(* Logix 5000 project; controller Receptivo vendor 1 type 14 code 106 rev 30.11; software revision 30.00; part 6 of 10 *)
(* tags used below, declared in another part *)
   Codigo_QAD3_Espacios : DINT;
   Codigo_QAD4_Espacios : DINT;
   Descripcion3_Espacios : DINT;
   Descripcion4_Espacios : DINT;
   Numero_Espacios_Descripcion_3 : DINT;
   Numero_Espacios_Descripcion_4 : DINT;
   Numero_Espacios_QAD3 : DINT;
   Numero_Espacios_QAD4 : DINT;
   Print3_Ejecute : BOOL;
   Print3_OK : BOOL;
   Print4_Ejecute : BOOL;
   Print4_OK : BOOL;
   CAJAS_3 : DINT;
   CAJAS_4 : DINT;
   Calendario : Hora_y_Fecha;
   CERO : DINT;
   Clima_3 : DINT;
   Clima_4 : DINT;
   Consecutivo : INT;
   Densidad_3 : REAL;
   Densidad_4 : REAL;
   Densidad_Bidon : REAL;
   Densidad_Bidon_1 : REAL;
   Densidad_Elmar_1 : REAL;
   Densidad_Fogg1_1 : REAL;
   Densidad_Fogg2_1 : REAL;
   EAN14_3 : Codigo_Barras;
   EAN14_4 : Codigo_Barras;
   Espacios : STRING;
   Estacion_1_GCola_1 : UDT_COLA;
   Estacion_1_General : UDT_GENERAL;
   Estacion_2_GCola_1 : UDT_COLA;
   ESTACION_3 : DINT;
   Estacion_3_GCola_1 : UDT_COLA;
   Estacion_3_General : UDT_GENERAL;
   Estacion_3_String : STRING;
   ESTACION_4 : DINT;
   Estacion_4_GCola_1 : UDT_COLA;
   Estacion_4_General : UDT_GENERAL;
   Estacion_4_String : STRING;
   LInea_General_3 : INT;
   LInea_General_4 : INT;
   Linea_String_General : STRING;
   Lote : DINT;
   Operador_3 : DINT;
   Operador_4 : DINT;
   Pesaje_3 : REAL;
   Pesaje_4 : REAL;
   Peso_Bidones : REAL;
   Peso_Bidones_1 : REAL;
   Peso_Caja_Elmar_1 : REAL;
   Peso_Caja_Fogg1_1 : REAL;
   Peso_Caja_Fogg2_1 : REAL;
   PESO_REAL_3 : DINT;
   PESO_REAL_4 : DINT;
   PESO_TEORICO_3 : DINT;
   PESO_TEORICO_4 : DINT;
   Producido_Bidones_Ahora : UDT_Maestro;
   Producido_Elmar_Ahora : UDT_Maestro;
   Producido_Fogg1_Ahora : UDT_Maestro;
   Producido_Fogg2_Ahora : UDT_Maestro;
   Producto3 : UDT_Inventario;
   Producto4 : UDT_Inventario;
   QAD_3 : STRING;
   QAD_4 : STRING;
   QAD_Auxiliar_Est4 : STRING;
(* MainProgram, continued *)

ROUTINE Estacion_3_Datos   (* ladder *)
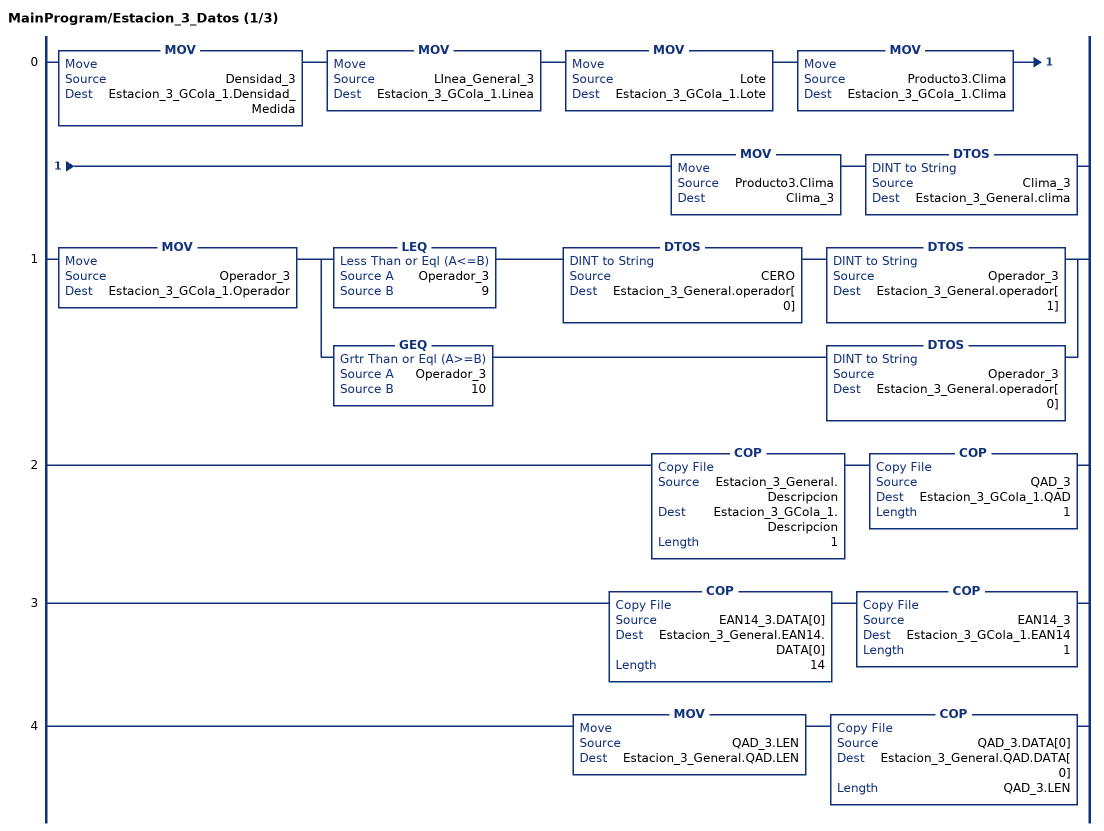
   0: MOV(Densidad_3,Estacion_3_GCola_1.Densidad_Medida)MOV(LInea_General_3,Estacion_3_GCola_1.Linea)MOV(Lote,Estacion_3_GCola_1.Lote)MOV(Producto3.Clima,Estacion_3_GCola_1.Clima)MOV(Producto3.Clima,Clima_3)DTOS(Clima_3,Estacion_3_General.clima);
   1: MOV(Operador_3,Estacion_3_GCola_1.Operador)[LEQ(Operador_3,9) DTOS(CERO,Estacion_3_General.operador[0]) DTOS(Operador_3,Estacion_3_General.operador[1]) ,GEQ(Operador_3,10) DTOS(Operador_3,Estacion_3_General.operador[0]) ];
   2: COP(Estacion_3_General.Descripcion,Estacion_3_GCola_1.Descripcion,1)COP(QAD_3,Estacion_3_GCola_1.QAD,1);
   3: COP(EAN14_3.DATA[0],Estacion_3_General.EAN14.DATA[0],14)COP(EAN14_3,Estacion_3_GCola_1.EAN14,1);
   4: MOV(QAD_3.LEN,Estacion_3_General.QAD.LEN)COP(QAD_3.DATA[0],Estacion_3_General.QAD.DATA[0],QAD_3.LEN);
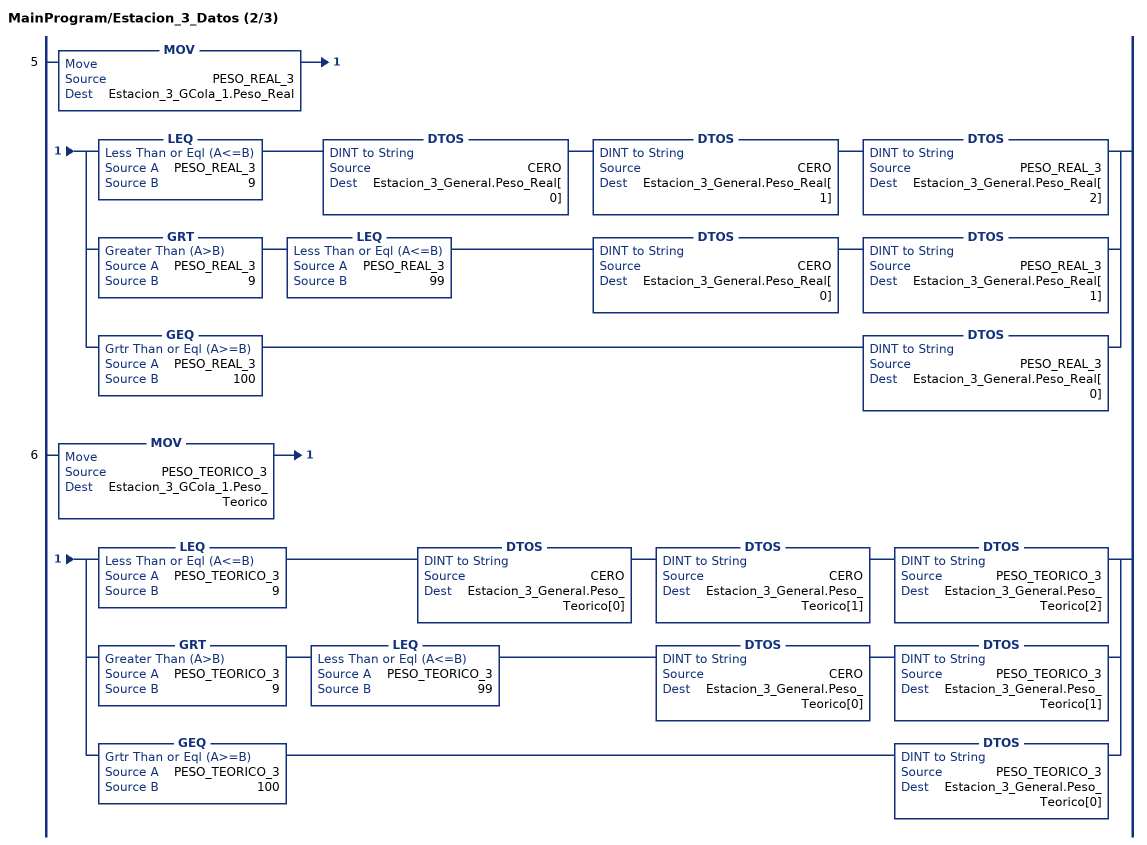
   5: MOV(PESO_REAL_3,Estacion_3_GCola_1.Peso_Real)[LEQ(PESO_REAL_3,9) DTOS(CERO,Estacion_3_General.Peso_Real[0]) DTOS(CERO,Estacion_3_General.Peso_Real[1]) DTOS(PESO_REAL_3,Estacion_3_General.Peso_Real[2]) ,GRT(PESO_REAL_3,9) LEQ(PESO_REAL_3,99) DTOS(CERO,Estacion_3_General.Peso_Real[0]) DTOS(PESO_REAL_3,Estacion_3_General.Peso_Real[1]) ,GEQ(PESO_REAL_3,100) DTOS(PESO_REAL_3,Estacion_3_General.Peso_Real[0]) ];
   6: MOV(PESO_TEORICO_3,Estacion_3_GCola_1.Peso_Teorico)[LEQ(PESO_TEORICO_3,9) DTOS(CERO,Estacion_3_General.Peso_Teorico[0]) DTOS(CERO,Estacion_3_General.Peso_Teorico[1]) DTOS(PESO_TEORICO_3,Estacion_3_General.Peso_Teorico[2]) ,GRT(PESO_TEORICO_3,9) LEQ(PESO_TEORICO_3,99) DTOS(CERO,Estacion_3_General.Peso_Teorico[0]) DTOS(PESO_TEORICO_3,Estacion_3_General.Peso_Teorico[1]) ,GEQ(PESO_TEORICO_3,100) DTOS(PESO_TEORICO_3,Estacion_3_General.Peso_Teorico[0]) ];
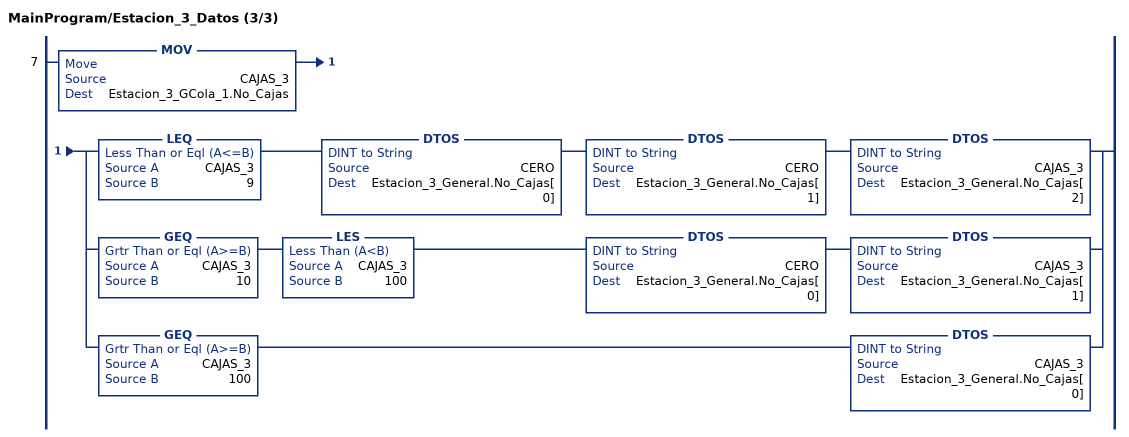
   7: MOV(CAJAS_3,Estacion_3_GCola_1.No_Cajas)[LEQ(CAJAS_3,9) DTOS(CERO,Estacion_3_General.No_Cajas[0]) DTOS(CERO,Estacion_3_General.No_Cajas[1]) DTOS(CAJAS_3,Estacion_3_General.No_Cajas[2]) ,GEQ(CAJAS_3,10) LES(CAJAS_3,100) DTOS(CERO,Estacion_3_General.No_Cajas[0]) DTOS(CAJAS_3,Estacion_3_General.No_Cajas[1]) ,GEQ(CAJAS_3,100) DTOS(CAJAS_3,Estacion_3_General.No_Cajas[0]) ];
END_ROUTINE

ROUTINE Estacion_3_To_Printer   (* ladder *)
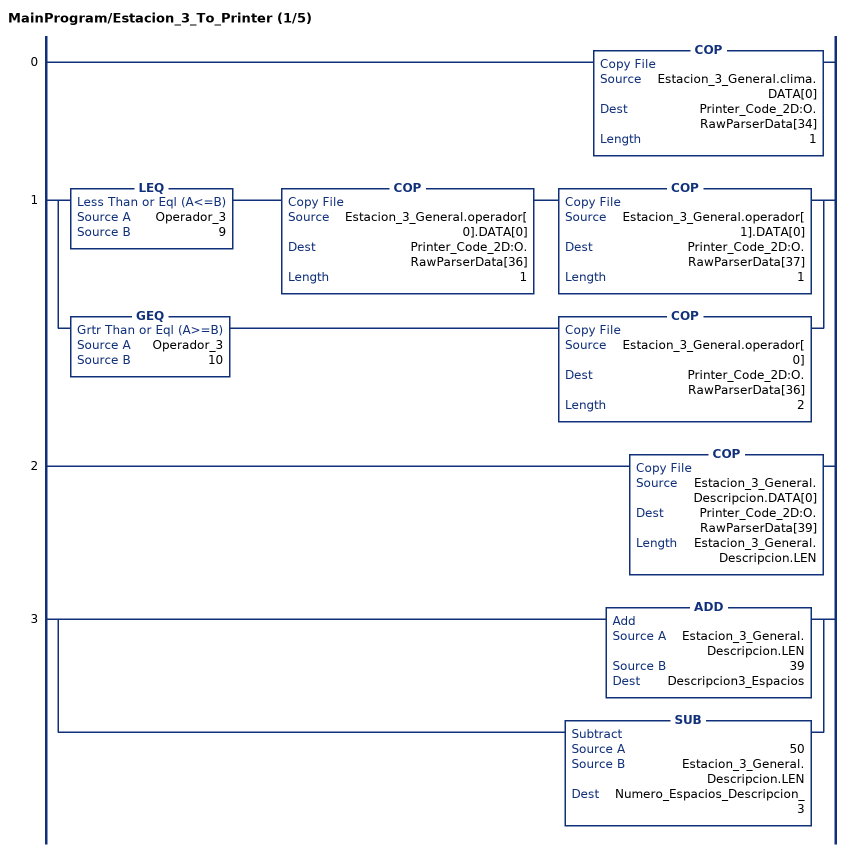
   0: COP(Estacion_3_General.clima.DATA[0],Printer_Code_2D:O.RawParserData[34],1);
   1: [LEQ(Operador_3,9) COP(Estacion_3_General.operador[0].DATA[0],Printer_Code_2D:O.RawParserData[36],1) COP(Estacion_3_General.operador[1].DATA[0],Printer_Code_2D:O.RawParserData[37],1) ,GEQ(Operador_3,10) COP(Estacion_3_General.operador[0],Printer_Code_2D:O.RawParserData[36],2) ];
   2: COP(Estacion_3_General.Descripcion.DATA[0],Printer_Code_2D:O.RawParserData[39],Estacion_3_General.Descripcion.LEN);
   3: [ADD(Estacion_3_General.Descripcion.LEN,39,Descripcion3_Espacios) ,SUB(50,Estacion_3_General.Descripcion.LEN,Numero_Espacios_Descripcion_3) ];
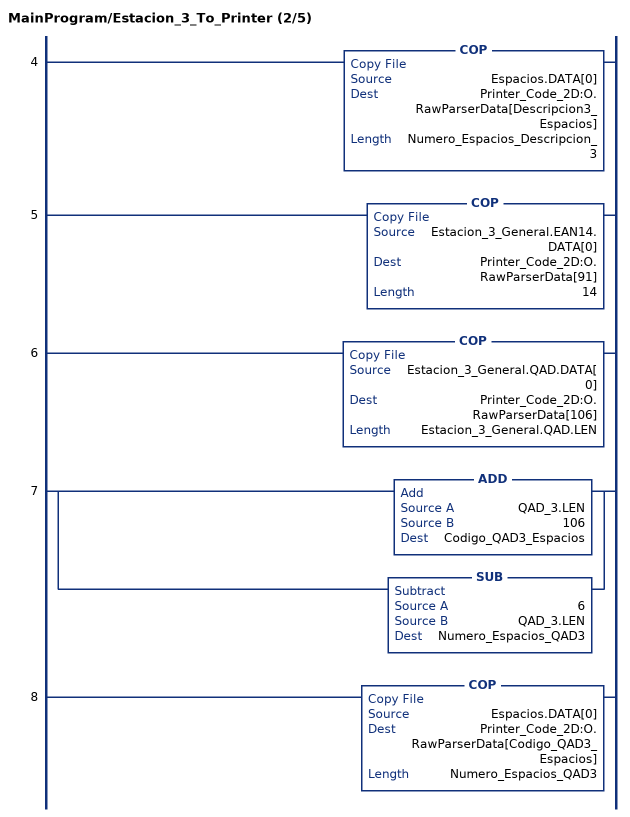
   4: COP(Espacios.DATA[0],Printer_Code_2D:O.RawParserData[Descripcion3_Espacios],Numero_Espacios_Descripcion_3);
   5: COP(Estacion_3_General.EAN14.DATA[0],Printer_Code_2D:O.RawParserData[91],14);
   6: COP(Estacion_3_General.QAD.DATA[0],Printer_Code_2D:O.RawParserData[106],Estacion_3_General.QAD.LEN);
   7: [ADD(QAD_3.LEN,106,Codigo_QAD3_Espacios) ,SUB(6,QAD_3.LEN,Numero_Espacios_QAD3) ];
   8: COP(Espacios.DATA[0],Printer_Code_2D:O.RawParserData[Codigo_QAD3_Espacios],Numero_Espacios_QAD3);
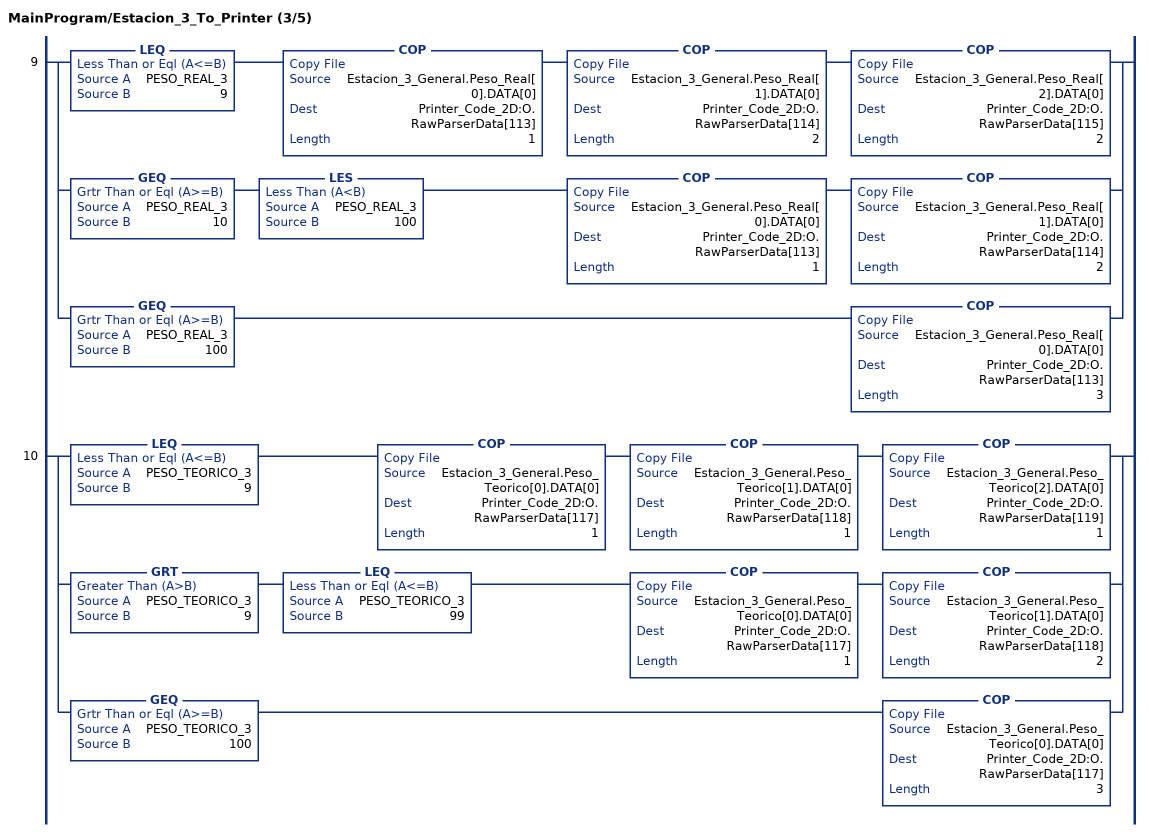
   9: [LEQ(PESO_REAL_3,9) COP(Estacion_3_General.Peso_Real[0].DATA[0],Printer_Code_2D:O.RawParserData[113],1) COP(Estacion_3_General.Peso_Real[1].DATA[0],Printer_Code_2D:O.RawParserData[114],2) COP(Estacion_3_General.Peso_Real[2].DATA[0],Printer_Code_2D:O.RawParserData[115],2) ,GEQ(PESO_REAL_3,10) LES(PESO_REAL_3,100) COP(Estacion_3_General.Peso_Real[0].DATA[0],Printer_Code_2D:O.RawParserData[113],1) COP(Estacion_3_General.Peso_Real[1].DATA[0],Printer_Code_2D:O.RawParserData[114],2) ,GEQ(PESO_REAL_3,100) COP(Estacion_3_General.Peso_Real[0].DATA[0],Printer_Code_2D:O.RawParserData[113],3) ];
   10: [LEQ(PESO_TEORICO_3,9) COP(Estacion_3_General.Peso_Teorico[0].DATA[0],Printer_Code_2D:O.RawParserData[117],1) COP(Estacion_3_General.Peso_Teorico[1].DATA[0],Printer_Code_2D:O.RawParserData[118],1) COP(Estacion_3_General.Peso_Teorico[2].DATA[0],Printer_Code_2D:O.RawParserData[119],1) ,GRT(PESO_TEORICO_3,9) LEQ(PESO_TEORICO_3,99) COP(Estacion_3_General.Peso_Teorico[0].DATA[0],Printer_Code_2D:O.RawParserData[117],1) COP(Estacion_3_General.Peso_Teorico[1].DATA[0],Printer_Code_2D:O.RawParserData[118],2) ,GEQ(PESO_TEORICO_3,100) COP(Estacion_3_General.Peso_Teorico[0].DATA[0],Printer_Code_2D:O.RawParserData[117],3) ];
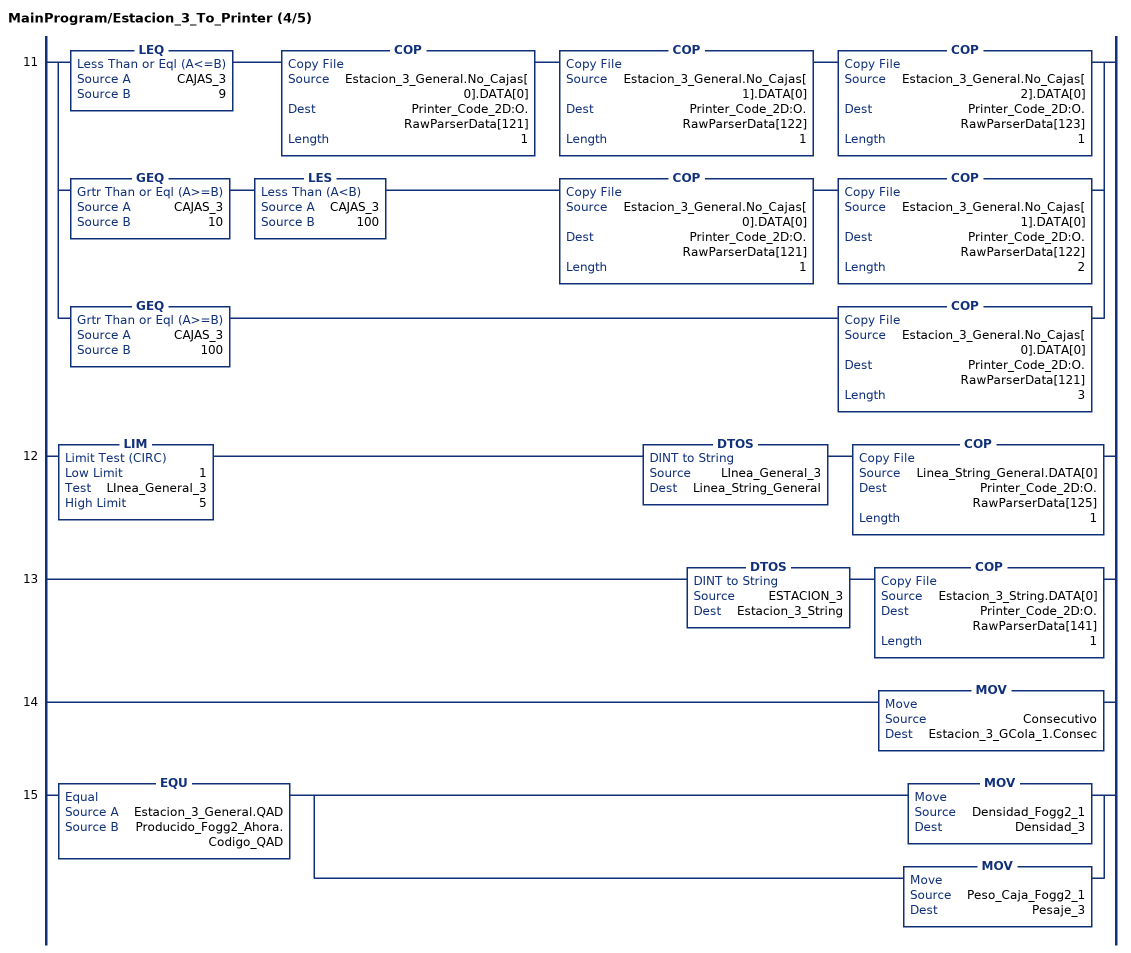
   11: [LEQ(CAJAS_3,9) COP(Estacion_3_General.No_Cajas[0].DATA[0],Printer_Code_2D:O.RawParserData[121],1) COP(Estacion_3_General.No_Cajas[1].DATA[0],Printer_Code_2D:O.RawParserData[122],1) COP(Estacion_3_General.No_Cajas[2].DATA[0],Printer_Code_2D:O.RawParserData[123],1) ,GEQ(CAJAS_3,10) LES(CAJAS_3,100) COP(Estacion_3_General.No_Cajas[0].DATA[0],Printer_Code_2D:O.RawParserData[121],1) COP(Estacion_3_General.No_Cajas[1].DATA[0],Printer_Code_2D:O.RawParserData[122],2) ,GEQ(CAJAS_3,100) COP(Estacion_3_General.No_Cajas[0].DATA[0],Printer_Code_2D:O.RawParserData[121],3) ];
   12: LIM(1,LInea_General_3,5)DTOS(LInea_General_3,Linea_String_General)COP(Linea_String_General.DATA[0],Printer_Code_2D:O.RawParserData[125],1);
   13: DTOS(ESTACION_3,Estacion_3_String)COP(Estacion_3_String.DATA[0],Printer_Code_2D:O.RawParserData[141],1);
   14: MOV(Consecutivo,Estacion_3_GCola_1.Consec);
   15: EQU(Estacion_3_General.QAD,Producido_Fogg2_Ahora.Codigo_QAD)[MOV(Densidad_Fogg2_1,Densidad_3) ,MOV(Peso_Caja_Fogg2_1,Pesaje_3) ];
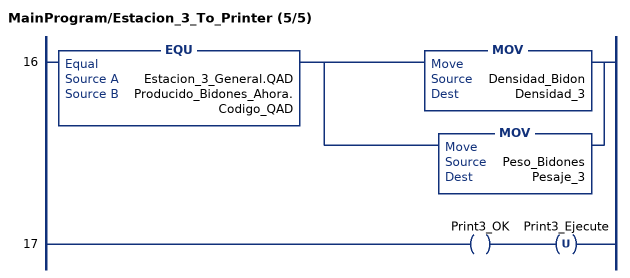
   16: EQU(Estacion_3_General.QAD,Producido_Bidones_Ahora.Codigo_QAD)[MOV(Densidad_Bidon,Densidad_3) ,MOV(Peso_Bidones,Pesaje_3) ];
   17: OTE(Print3_OK)OTU(Print3_Ejecute);
END_ROUTINE

ROUTINE Estacion_4_Datos   (* ladder *)
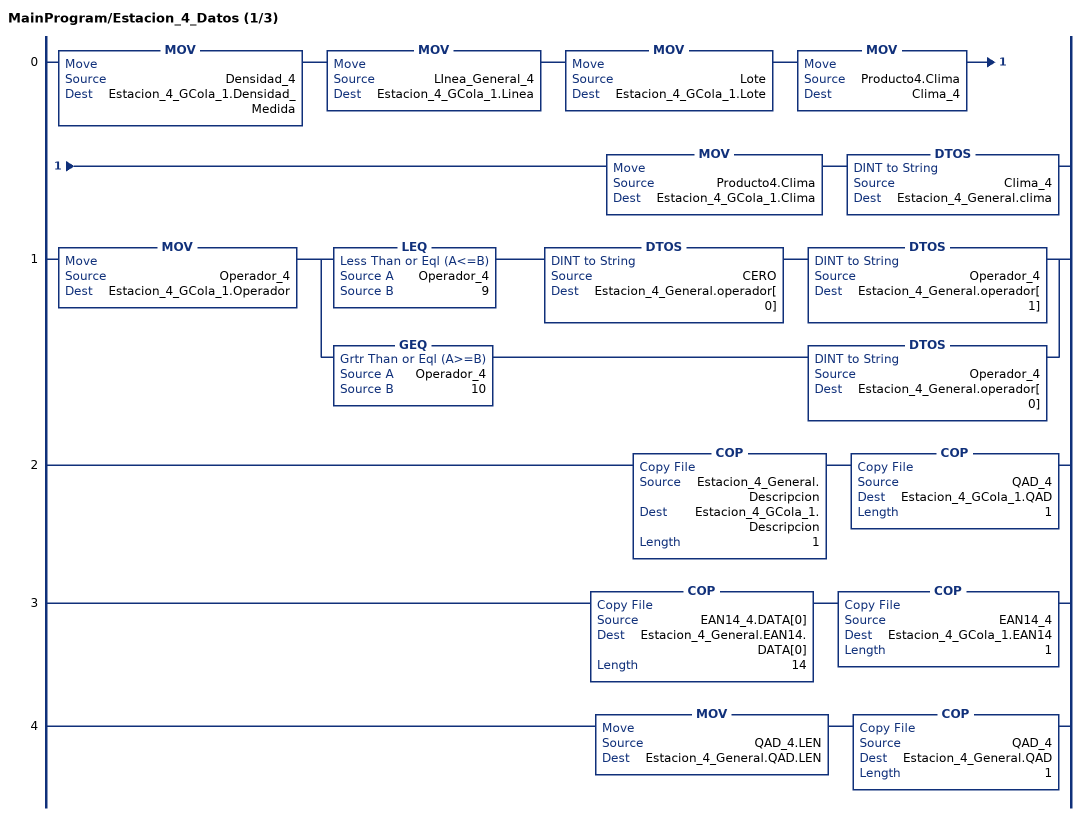
   0: MOV(Densidad_4,Estacion_4_GCola_1.Densidad_Medida)MOV(LInea_General_4,Estacion_4_GCola_1.Linea)MOV(Lote,Estacion_4_GCola_1.Lote)MOV(Producto4.Clima,Clima_4)MOV(Producto4.Clima,Estacion_4_GCola_1.Clima)DTOS(Clima_4,Estacion_4_General.clima);
   1: MOV(Operador_4,Estacion_4_GCola_1.Operador)[LEQ(Operador_4,9) DTOS(CERO,Estacion_4_General.operador[0]) DTOS(Operador_4,Estacion_4_General.operador[1]) ,GEQ(Operador_4,10) DTOS(Operador_4,Estacion_4_General.operador[0]) ];
   2: COP(Estacion_4_General.Descripcion,Estacion_4_GCola_1.Descripcion,1)COP(QAD_4,Estacion_4_GCola_1.QAD,1);
   3: COP(EAN14_4.DATA[0],Estacion_4_General.EAN14.DATA[0],14)COP(EAN14_4,Estacion_4_GCola_1.EAN14,1);
   4: MOV(QAD_4.LEN,Estacion_4_General.QAD.LEN)COP(QAD_4,Estacion_4_General.QAD,1);
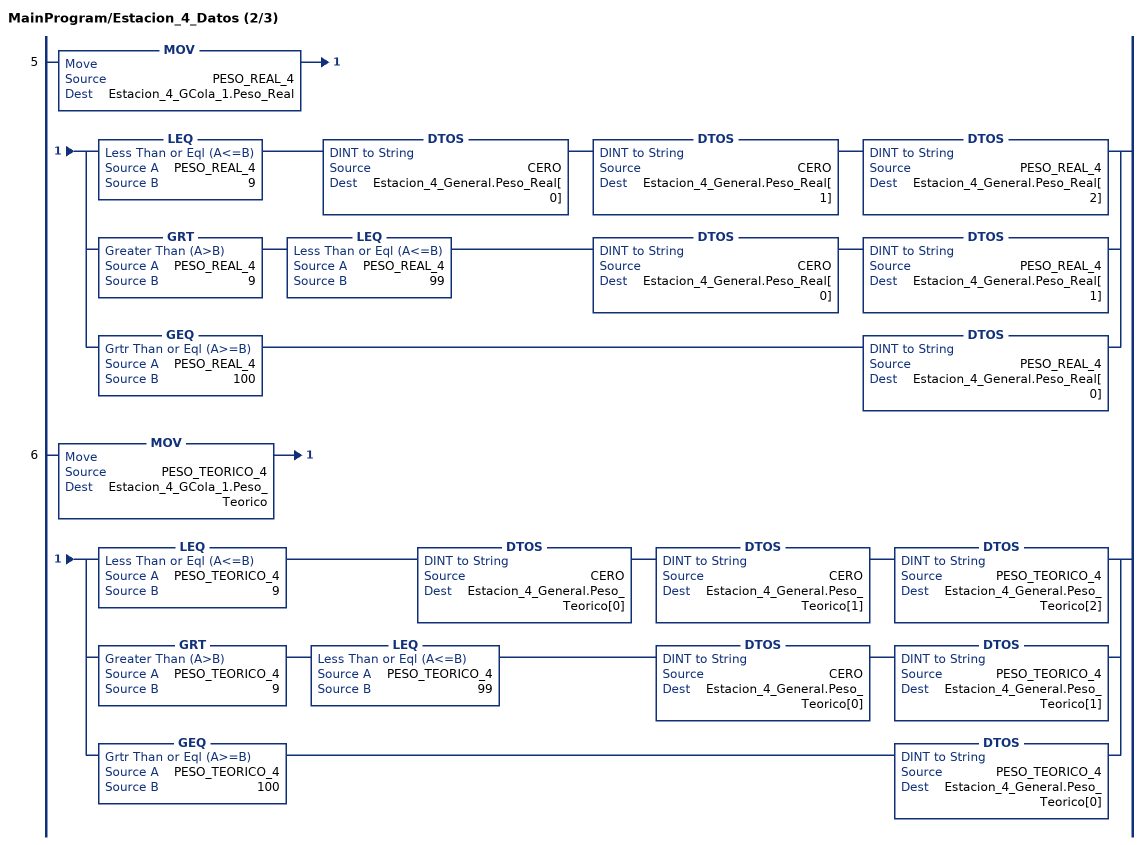
   5: MOV(PESO_REAL_4,Estacion_4_GCola_1.Peso_Real)[LEQ(PESO_REAL_4,9) DTOS(CERO,Estacion_4_General.Peso_Real[0]) DTOS(CERO,Estacion_4_General.Peso_Real[1]) DTOS(PESO_REAL_4,Estacion_4_General.Peso_Real[2]) ,GRT(PESO_REAL_4,9) LEQ(PESO_REAL_4,99) DTOS(CERO,Estacion_4_General.Peso_Real[0]) DTOS(PESO_REAL_4,Estacion_4_General.Peso_Real[1]) ,GEQ(PESO_REAL_4,100) DTOS(PESO_REAL_4,Estacion_4_General.Peso_Real[0]) ];
   6: MOV(PESO_TEORICO_4,Estacion_4_GCola_1.Peso_Teorico)[LEQ(PESO_TEORICO_4,9) DTOS(CERO,Estacion_4_General.Peso_Teorico[0]) DTOS(CERO,Estacion_4_General.Peso_Teorico[1]) DTOS(PESO_TEORICO_4,Estacion_4_General.Peso_Teorico[2]) ,GRT(PESO_TEORICO_4,9) LEQ(PESO_TEORICO_4,99) DTOS(CERO,Estacion_4_General.Peso_Teorico[0]) DTOS(PESO_TEORICO_4,Estacion_4_General.Peso_Teorico[1]) ,GEQ(PESO_TEORICO_4,100) DTOS(PESO_TEORICO_4,Estacion_4_General.Peso_Teorico[0]) ];
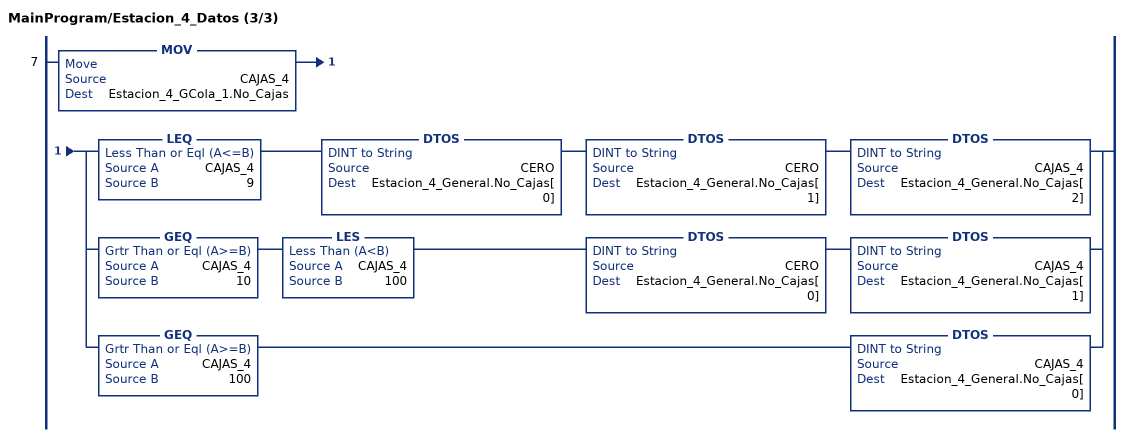
   7: MOV(CAJAS_4,Estacion_4_GCola_1.No_Cajas)[LEQ(CAJAS_4,9) DTOS(CERO,Estacion_4_General.No_Cajas[0]) DTOS(CERO,Estacion_4_General.No_Cajas[1]) DTOS(CAJAS_4,Estacion_4_General.No_Cajas[2]) ,GEQ(CAJAS_4,10) LES(CAJAS_4,100) DTOS(CERO,Estacion_4_General.No_Cajas[0]) DTOS(CAJAS_4,Estacion_4_General.No_Cajas[1]) ,GEQ(CAJAS_4,100) DTOS(CAJAS_4,Estacion_4_General.No_Cajas[0]) ];
END_ROUTINE

ROUTINE Estacion_4_To_Printer   (* ladder *)
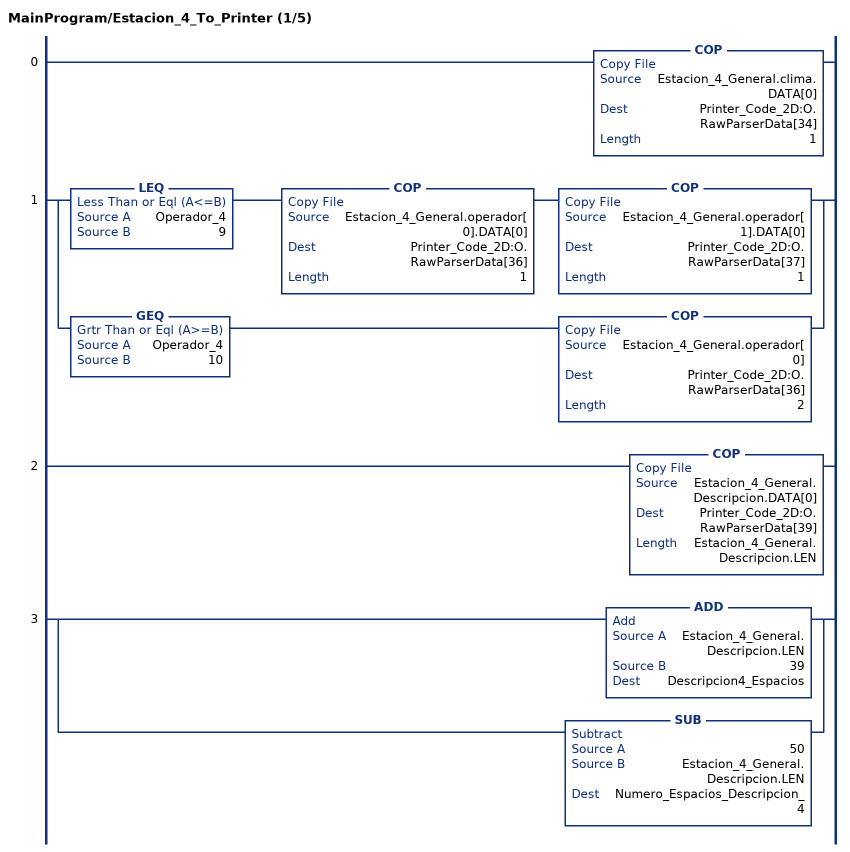
   0: COP(Estacion_4_General.clima.DATA[0],Printer_Code_2D:O.RawParserData[34],1);
   1: [LEQ(Operador_4,9) COP(Estacion_4_General.operador[0].DATA[0],Printer_Code_2D:O.RawParserData[36],1) COP(Estacion_4_General.operador[1].DATA[0],Printer_Code_2D:O.RawParserData[37],1) ,GEQ(Operador_4,10) COP(Estacion_4_General.operador[0],Printer_Code_2D:O.RawParserData[36],2) ];
   2: COP(Estacion_4_General.Descripcion.DATA[0],Printer_Code_2D:O.RawParserData[39],Estacion_4_General.Descripcion.LEN);
   3: [ADD(Estacion_4_General.Descripcion.LEN,39,Descripcion4_Espacios) ,SUB(50,Estacion_4_General.Descripcion.LEN,Numero_Espacios_Descripcion_4) ];
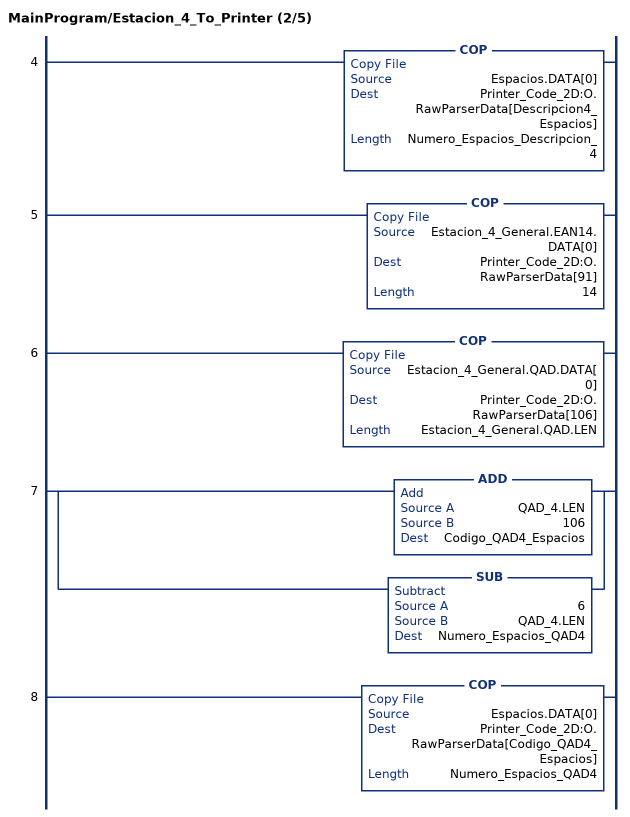
   4: COP(Espacios.DATA[0],Printer_Code_2D:O.RawParserData[Descripcion4_Espacios],Numero_Espacios_Descripcion_4);
   5: COP(Estacion_4_General.EAN14.DATA[0],Printer_Code_2D:O.RawParserData[91],14);
   6: COP(Estacion_4_General.QAD.DATA[0],Printer_Code_2D:O.RawParserData[106],Estacion_4_General.QAD.LEN);
   7: [ADD(QAD_4.LEN,106,Codigo_QAD4_Espacios) ,SUB(6,QAD_4.LEN,Numero_Espacios_QAD4) ];
   8: COP(Espacios.DATA[0],Printer_Code_2D:O.RawParserData[Codigo_QAD4_Espacios],Numero_Espacios_QAD4);
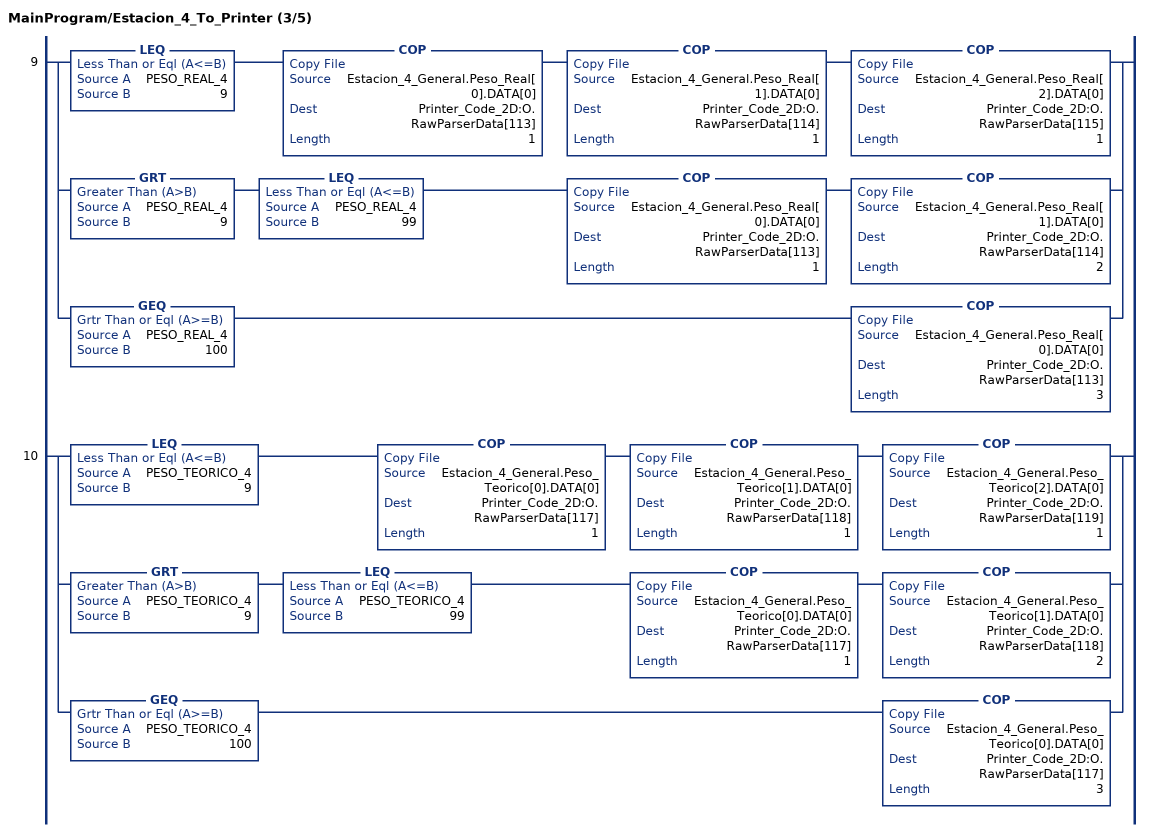
   9: [LEQ(PESO_REAL_4,9) COP(Estacion_4_General.Peso_Real[0].DATA[0],Printer_Code_2D:O.RawParserData[113],1) COP(Estacion_4_General.Peso_Real[1].DATA[0],Printer_Code_2D:O.RawParserData[114],1) COP(Estacion_4_General.Peso_Real[2].DATA[0],Printer_Code_2D:O.RawParserData[115],1) ,GRT(PESO_REAL_4,9) LEQ(PESO_REAL_4,99) COP(Estacion_4_General.Peso_Real[0].DATA[0],Printer_Code_2D:O.RawParserData[113],1) COP(Estacion_4_General.Peso_Real[1].DATA[0],Printer_Code_2D:O.RawParserData[114],2) ,GEQ(PESO_REAL_4,100) COP(Estacion_4_General.Peso_Real[0].DATA[0],Printer_Code_2D:O.RawParserData[113],3) ];
   10: [LEQ(PESO_TEORICO_4,9) COP(Estacion_4_General.Peso_Teorico[0].DATA[0],Printer_Code_2D:O.RawParserData[117],1) COP(Estacion_4_General.Peso_Teorico[1].DATA[0],Printer_Code_2D:O.RawParserData[118],1) COP(Estacion_4_General.Peso_Teorico[2].DATA[0],Printer_Code_2D:O.RawParserData[119],1) ,GRT(PESO_TEORICO_4,9) LEQ(PESO_TEORICO_4,99) COP(Estacion_4_General.Peso_Teorico[0].DATA[0],Printer_Code_2D:O.RawParserData[117],1) COP(Estacion_4_General.Peso_Teorico[1].DATA[0],Printer_Code_2D:O.RawParserData[118],2) ,GEQ(PESO_TEORICO_4,100) COP(Estacion_4_General.Peso_Teorico[0].DATA[0],Printer_Code_2D:O.RawParserData[117],3) ];
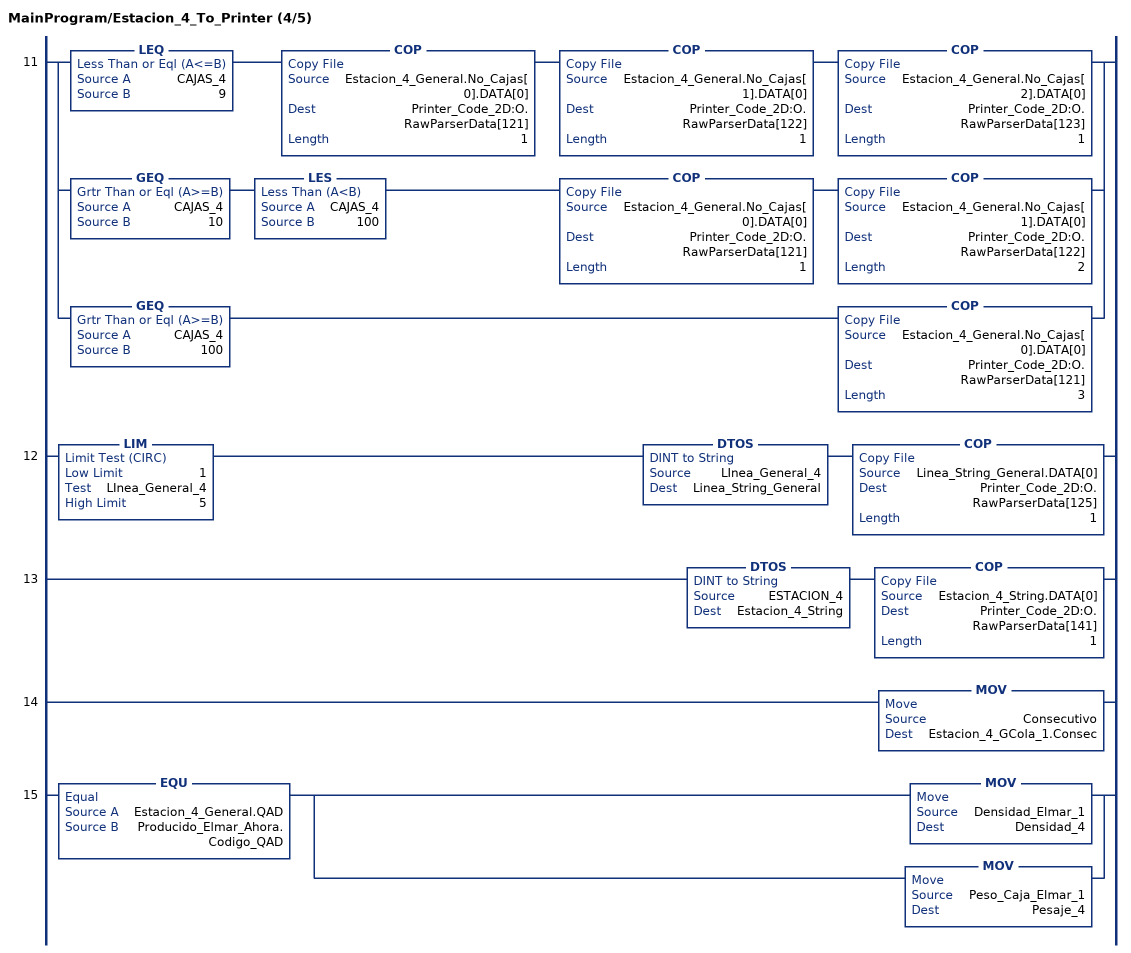
   11: [LEQ(CAJAS_4,9) COP(Estacion_4_General.No_Cajas[0].DATA[0],Printer_Code_2D:O.RawParserData[121],1) COP(Estacion_4_General.No_Cajas[1].DATA[0],Printer_Code_2D:O.RawParserData[122],1) COP(Estacion_4_General.No_Cajas[2].DATA[0],Printer_Code_2D:O.RawParserData[123],1) ,GEQ(CAJAS_4,10) LES(CAJAS_4,100) COP(Estacion_4_General.No_Cajas[0].DATA[0],Printer_Code_2D:O.RawParserData[121],1) COP(Estacion_4_General.No_Cajas[1].DATA[0],Printer_Code_2D:O.RawParserData[122],2) ,GEQ(CAJAS_4,100) COP(Estacion_4_General.No_Cajas[0].DATA[0],Printer_Code_2D:O.RawParserData[121],3) ];
   12: LIM(1,LInea_General_4,5)DTOS(LInea_General_4,Linea_String_General)COP(Linea_String_General.DATA[0],Printer_Code_2D:O.RawParserData[125],1);
   13: DTOS(ESTACION_4,Estacion_4_String)COP(Estacion_4_String.DATA[0],Printer_Code_2D:O.RawParserData[141],1);
   14: MOV(Consecutivo,Estacion_4_GCola_1.Consec);
   15: EQU(Estacion_4_General.QAD,Producido_Elmar_Ahora.Codigo_QAD)[MOV(Densidad_Elmar_1,Densidad_4) ,MOV(Peso_Caja_Elmar_1,Pesaje_4) ];
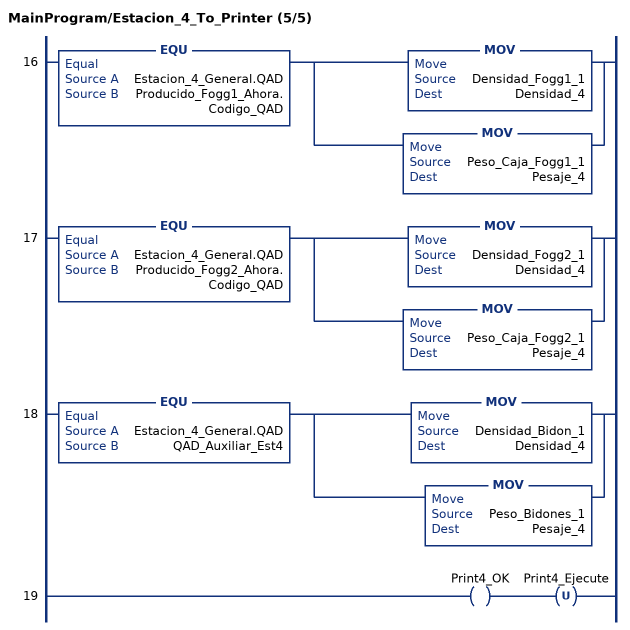
   16: EQU(Estacion_4_General.QAD,Producido_Fogg1_Ahora.Codigo_QAD)[MOV(Densidad_Fogg1_1,Densidad_4) ,MOV(Peso_Caja_Fogg1_1,Pesaje_4) ];
   17: EQU(Estacion_4_General.QAD,Producido_Fogg2_Ahora.Codigo_QAD)[MOV(Densidad_Fogg2_1,Densidad_4) ,MOV(Peso_Caja_Fogg2_1,Pesaje_4) ];
   18: EQU(Estacion_4_General.QAD,QAD_Auxiliar_Est4)[MOV(Densidad_Bidon_1,Densidad_4) ,MOV(Peso_Bidones_1,Pesaje_4) ];
   19: OTE(Print4_OK)OTU(Print4_Ejecute);
END_ROUTINE

ROUTINE Get_Date_Time   (* ladder *)
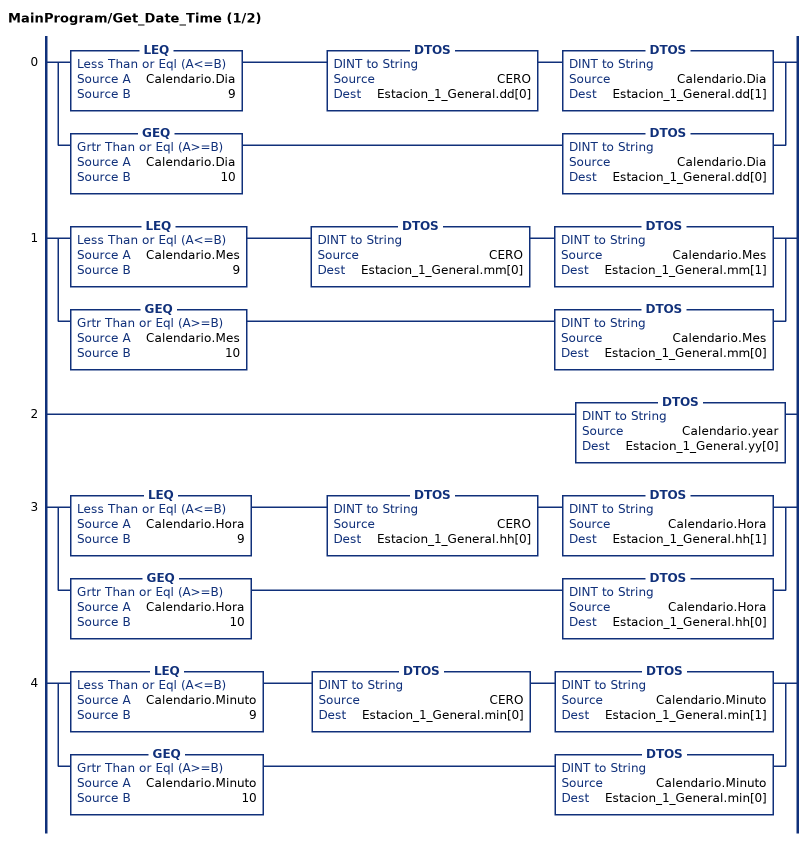
   0: [LEQ(Calendario.Dia,9) DTOS(CERO,Estacion_1_General.dd[0]) DTOS(Calendario.Dia,Estacion_1_General.dd[1]) ,GEQ(Calendario.Dia,10) DTOS(Calendario.Dia,Estacion_1_General.dd[0]) ];
   1: [LEQ(Calendario.Mes,9) DTOS(CERO,Estacion_1_General.mm[0]) DTOS(Calendario.Mes,Estacion_1_General.mm[1]) ,GEQ(Calendario.Mes,10) DTOS(Calendario.Mes,Estacion_1_General.mm[0]) ];
   2: DTOS(Calendario.year,Estacion_1_General.yy[0]);
   3: [LEQ(Calendario.Hora,9) DTOS(CERO,Estacion_1_General.hh[0]) DTOS(Calendario.Hora,Estacion_1_General.hh[1]) ,GEQ(Calendario.Hora,10) DTOS(Calendario.Hora,Estacion_1_General.hh[0]) ];
   4: [LEQ(Calendario.Minuto,9) DTOS(CERO,Estacion_1_General.min[0]) DTOS(Calendario.Minuto,Estacion_1_General.min[1]) ,GEQ(Calendario.Minuto,10) DTOS(Calendario.Minuto,Estacion_1_General.min[0]) ];
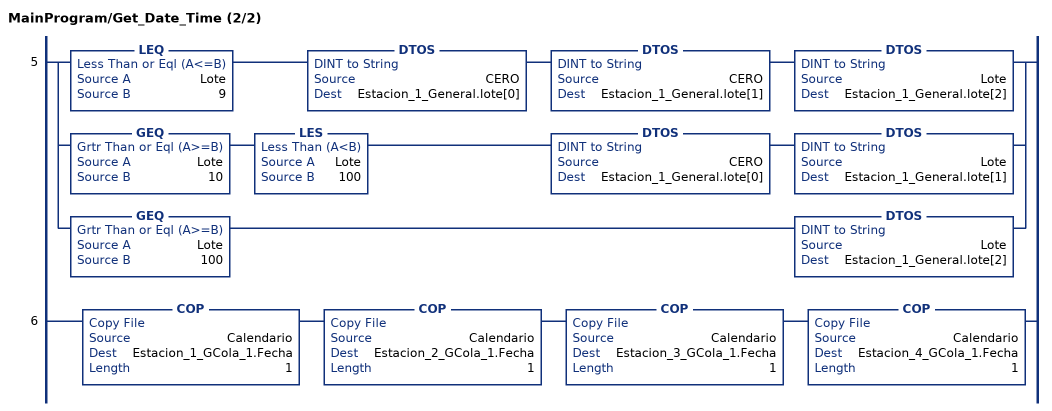
   5: [LEQ(Lote,9) DTOS(CERO,Estacion_1_General.lote[0]) DTOS(CERO,Estacion_1_General.lote[1]) DTOS(Lote,Estacion_1_General.lote[2]) ,GEQ(Lote,10) LES(Lote,100) DTOS(CERO,Estacion_1_General.lote[0]) DTOS(Lote,Estacion_1_General.lote[1]) ,GEQ(Lote,100) DTOS(Lote,Estacion_1_General.lote[2]) ];
   6: COP(Calendario,Estacion_1_GCola_1.Fecha,1)COP(Calendario,Estacion_2_GCola_1.Fecha,1)COP(Calendario,Estacion_3_GCola_1.Fecha,1)COP(Calendario,Estacion_4_GCola_1.Fecha,1);
END_ROUTINE
